# EPICS substitutions: VCSIOCAG10/db/user.substitutions
# Example substitutions file

file "db/dbExample1.db" {
    { user = "yann" }
}

file db/dbExample2.db {
    pattern { user, no, scan }
        { "yann", 1, "1 second" }
        { "yann", 2, "2 second" }
        { "yann", 3, "5 second" }
}
